Fanuc KAREL source: ko00052.KL

-- PROVISIONAL review KL for V770-1; original PC SHA256 9c9671c46c4c6e72014e52a5c039d5b1e4b643295983a97632199e57268024a8
-- Incomplete behavior may be omitted. Consult companion uncertainty JSON. Do not deploy.
PROGRAM KO00052
%NOLOCKGROUP
BEGIN
  -- UNRESOLVED_PC offsets 5-12; opcodes 9D,23
  -- UNRESOLVED_PC offsets 17-66; opcodes 27,27,49,7E,AD,22,1C,22,31,7E,4A
  -- UNRESOLVED_PC offsets 71-75; opcodes 7F
END KO00052
